Fanuc KAREL source: kt00114.KL

-- PROVISIONAL review KL for V940-1; original PC SHA256 8447c851eba2876a4e721304ffc3794d411f85d9c301772c0b52be48f04a1cd8
-- Incomplete behavior may be omitted. Consult companion uncertainty JSON. Do not deploy.
PROGRAM KT00114
%NOLOCKGROUP
VAR
  I2 : INTEGER
  OUT : REAL
-- UNRESOLVED_DECL Y1 type=002018
BEGIN
  -- V9_ZERO_TABLE_METADATA_HINT layout=0001; no indexed target words; source/name/runtime held
  -- UNRESOLVED_PC offsets 5-19; opcodes 2E,22,9D,33,B2
  -- UNRESOLVED_PC offsets 24-35; opcodes 2E,23
  -- UNRESOLVED_PC offsets 40-66; opcodes 22,9D,33,B1,21,64,29,64,29,6C,23
  -- UNRESOLVED_PC offsets 71-75; opcodes 7F
END KT00114
